FUNCTION_BLOCK "Semantic_IecTimerInOutput"
{ S7_Optimized_Access := 'TRUE' }
VERSION : 0.1

VAR_OUTPUT
    badTimer : IEC_TIMER;
    // EXPECT: error[type.illegal-section] SEM-SECTION-004
END_VAR

BEGIN
END_FUNCTION_BLOCK
